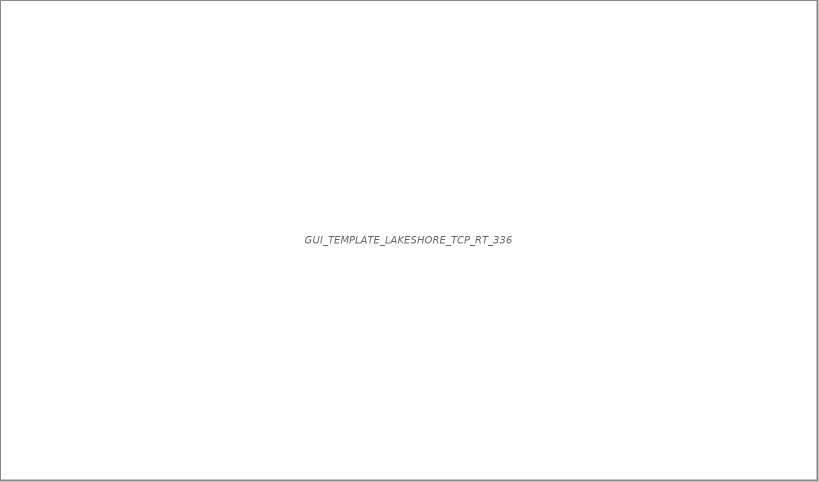
VISUALIZATION GUI_LAKESHORE_TCP_RT_336  // 819x482
    Frame (0,0 817x480)
        shows GUI_TEMPLATE_LAKESHORE_TCP_RT_336(m_Instance := MAIN.LS336_TCP_RT)
END_VISUALIZATION

(* stored: Version 1.1.0.1, ProductVersion 3.1.4022.16
   Visu GUI_LAKESHORE_TCP_RT_336: Id {dd9ea695-4aff-4c07-8a32-540a720a6857} *)
